// TIA Portal V20 export
FUNCTION_BLOCK "FB_Digital_Input"   // FB1, LAD
{ S7_Optimized_Access := 'TRUE' }
// stored: MemoryReserve 100, SetENOAutomatically false
   VAR_INPUT
      DI_Emergency_Stop_Release : Bool;
      DI_Sensor_Water_Fountain_Before_Entrace_Functional_Test_Spinner_Conveyor_Belt : Bool;
      DI_Sensor_Water_Fountain_Entrace_Functional_Test_Spinner_Conveyor_Belt : Bool;
      DI_Sensor_Water_Fountain_Entrace_Functional_Test_After_Spinner_Conveyor_Belt : Bool;
      DI_Trigger_Read_Serial_Number_Entrace_Functional_Test : Bool;
      DI_Sensor_Water_Fountain_Geting_Exit_Rework_Conveyor_Belt : Bool;
      DI_Button_Water_Fountain_Get_Exit_Rework_Conveyor_Belt : Bool;
      DI_Trigger_Read_Serial_Number_Exit_Functional_Test : Bool;
      DI_Sensor_Water_Fountain_Exit_Functional_Test_Spinner_Conveyor_Belt : Bool;
      DI_Sensor_Water_Fountain_Exit_Functional_Test_After_Spinner_Conveyor_Belt : Bool;
      DI_Sensor_Water_Fountain_Geting_Entrace_Rework_Conveyor_Belt_Start : Bool;
      DI_Sensor_Water_Fountain_Geting_Entrace_Rework_Conveyor_Belt_Finish : Bool;
      DI_Carousel_Frequency_Inverter_Fail : Bool;
      DI_Conveyor_Belt_Functional_Test_Inverter_Fail : Bool;
      DI_Selected_Voltage_220V : Bool;
      DI_Selected_Voltage_127V : Bool;
      DI_Sensor_Spinner_Entrace_Functional_Test_Position_Withdrawn : Bool;
      DI_Sensor_Spinner_Entrace_Functional_Test_Position_Advanced : Bool;
      DI_Sensor_Spinner_Exit_Functional_Test_Position_Withdrawn : Bool;
      DI_Sensor_Spinner_Exit_Functional_Test_Position_Advanced : Bool;
      DI_Digital_Input_20 : Bool;
      DI_Digital_Input_21 : Bool;
      DI_Digital_Input_22 : Bool;
      DI_Digital_Input_23 : Bool;
      DI_Digital_Input_24 : Bool;
      DI_Digital_Input_25 : Bool;
      DI_Digital_Input_26 : Bool;
      DI_Digital_Input_27 : Bool;
      DI_Digital_Input_28 : Bool;
      DI_Digital_Input_29 : Bool;
   END_VAR
   VAR_OUTPUT
      DB_Emergency_Stop_Release : Bool;
      DB_Sensor_Water_Fountain_Before_Entrace_Functional_Test_Spinner_Conveyor_Belt : Bool;
      DB_Sensor_Water_Fountain_Entrace_Functional_Test_Spinner_Conveyor_Belt : Bool;
      DB_Sensor_Water_Fountain_Entrace_Functional_Test_After_Spinner_Conveyor_Belt : Bool;
      DB_Trigger_Read_Serial_Number_Entrace_Functional_Test : Bool;
      DB_Sensor_Water_Fountain_Geting_Exit_Rework_Conveyor_Belt : Bool;
      DB_Button_Water_Fountain_Get_Exit_Rework_Conveyor_Belt : Bool;
      DB_Trigger_Read_Serial_Number_Exit_Functional_Test : Bool;
      DB_Sensor_Water_Fountain_Exit_Functional_Test_Spinner_Conveyor_Belt : Bool;
      DB_Sensor_Water_Fountain_Exit_Functional_Test_After_Spinner_Conveyor_Belt : Bool;
      DB_Sensor_Water_Fountain_Geting_Entrace_Rework_Conveyor_Belt_Start : Bool;
      DB_Sensor_Water_Fountain_Geting_Entrace_Rework_Conveyor_Belt_Finish : Bool;
      DB_Carousel_Frequency_Inverter_Fail : Bool;
      DB_Conveyor_Belt_Functional_Test_Inverter_Fail : Bool;
      DB_Selected_Voltage_220V : Bool;
      DB_Selected_Voltage_127V : Bool;
      DB_Sensor_Spinner_Entrace_Functional_Test_Position_Withdrawn : Bool;
      DB_Sensor_Spinner_Entrace_Functional_Test_Position_Advanced : Bool;
      DB_Sensor_Spinner_Exit_Functional_Test_Position_Withdrawn : Bool;
      DB_Sensor_Spinner_Exit_Functional_Test_Position_Advanced : Bool;
      DB_Digital_Input_20 : Bool;
      DB_Digital_Input_21 : Bool;
      DB_Digital_Input_22 : Bool;
      DB_Digital_Input_23 : Bool;
      DB_Digital_Input_24 : Bool;
      DB_Digital_Input_25 : Bool;
      DB_Digital_Input_26 : Bool;
      DB_Digital_Input_27 : Bool;
      DB_Digital_Input_28 : Bool;
      DB_Digital_Input_29 : Bool;
   END_VAR
BEGIN

REGION Network 1
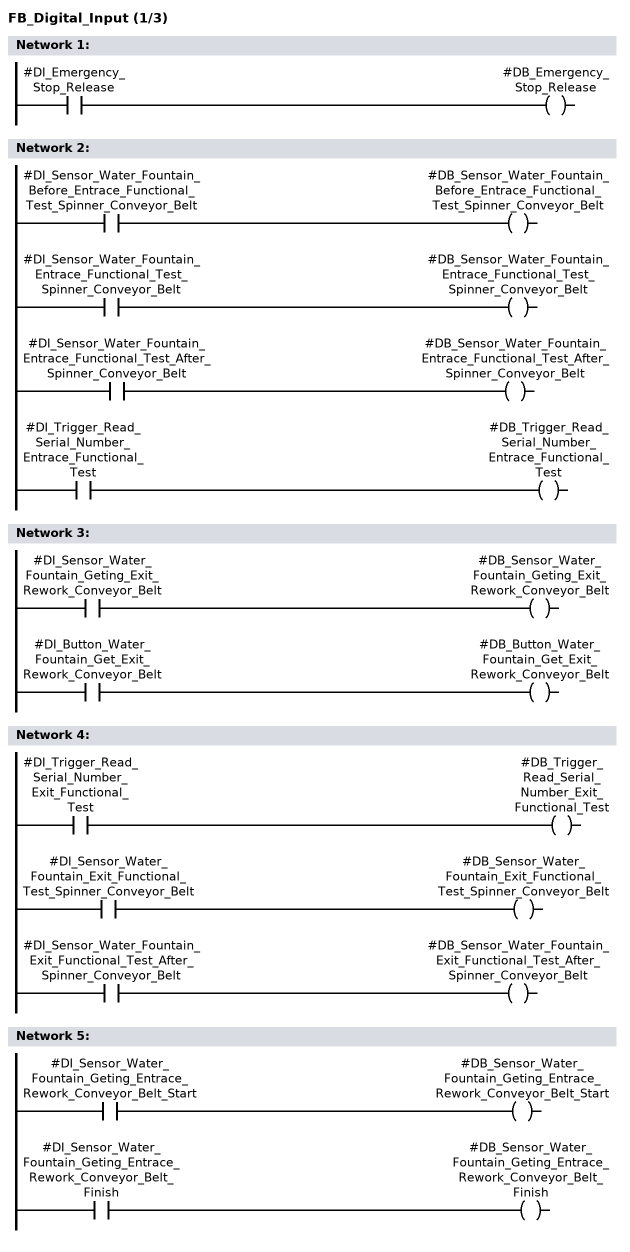
   RUNG wire#powerrail
      Contact( #DI_Emergency_Stop_Release )
      Coil( #DB_Emergency_Stop_Release )
   END_RUNG
   // the same network as SCL:
   #DB_Emergency_Stop_Release := #DI_Emergency_Stop_Release;
END_REGION

REGION Network 2
   RUNG wire#powerrail
      Contact( #DI_Sensor_Water_Fountain_Before_Entrace_Functional_Test_Spinner_Conveyor_Belt )
      Coil( #DB_Sensor_Water_Fountain_Before_Entrace_Functional_Test_Spinner_Conveyor_Belt )
   END_RUNG
   RUNG wire#powerrail
      Contact( #DI_Sensor_Water_Fountain_Entrace_Functional_Test_Spinner_Conveyor_Belt )
      Coil( #DB_Sensor_Water_Fountain_Entrace_Functional_Test_Spinner_Conveyor_Belt )
   END_RUNG
   RUNG wire#powerrail
      Contact( #DI_Sensor_Water_Fountain_Entrace_Functional_Test_After_Spinner_Conveyor_Belt )
      Coil( #DB_Sensor_Water_Fountain_Entrace_Functional_Test_After_Spinner_Conveyor_Belt )
   END_RUNG
   RUNG wire#powerrail
      Contact( #DI_Trigger_Read_Serial_Number_Entrace_Functional_Test )
      Coil( #DB_Trigger_Read_Serial_Number_Entrace_Functional_Test )
   END_RUNG
   // the same network as SCL:
   #DB_Sensor_Water_Fountain_Before_Entrace_Functional_Test_Spinner_Conveyor_Belt := #DI_Sensor_Water_Fountain_Before_Entrace_Functional_Test_Spinner_Conveyor_Belt;
   #DB_Sensor_Water_Fountain_Entrace_Functional_Test_Spinner_Conveyor_Belt := #DI_Sensor_Water_Fountain_Entrace_Functional_Test_Spinner_Conveyor_Belt;
   #DB_Sensor_Water_Fountain_Entrace_Functional_Test_After_Spinner_Conveyor_Belt := #DI_Sensor_Water_Fountain_Entrace_Functional_Test_After_Spinner_Conveyor_Belt;
   #DB_Trigger_Read_Serial_Number_Entrace_Functional_Test := #DI_Trigger_Read_Serial_Number_Entrace_Functional_Test;
END_REGION

REGION Network 3
   RUNG wire#powerrail
      Contact( #DI_Sensor_Water_Fountain_Geting_Exit_Rework_Conveyor_Belt )
      Coil( #DB_Sensor_Water_Fountain_Geting_Exit_Rework_Conveyor_Belt )
   END_RUNG
   RUNG wire#powerrail
      Contact( #DI_Button_Water_Fountain_Get_Exit_Rework_Conveyor_Belt )
      Coil( #DB_Button_Water_Fountain_Get_Exit_Rework_Conveyor_Belt )
   END_RUNG
   // the same network as SCL:
   #DB_Sensor_Water_Fountain_Geting_Exit_Rework_Conveyor_Belt := #DI_Sensor_Water_Fountain_Geting_Exit_Rework_Conveyor_Belt;
   #DB_Button_Water_Fountain_Get_Exit_Rework_Conveyor_Belt := #DI_Button_Water_Fountain_Get_Exit_Rework_Conveyor_Belt;
END_REGION

REGION Network 4
   RUNG wire#powerrail
      Contact( #DI_Trigger_Read_Serial_Number_Exit_Functional_Test )
      Coil( #DB_Trigger_Read_Serial_Number_Exit_Functional_Test )
   END_RUNG
   RUNG wire#powerrail
      Contact( #DI_Sensor_Water_Fountain_Exit_Functional_Test_Spinner_Conveyor_Belt )
      Coil( #DB_Sensor_Water_Fountain_Exit_Functional_Test_Spinner_Conveyor_Belt )
   END_RUNG
   RUNG wire#powerrail
      Contact( #DI_Sensor_Water_Fountain_Exit_Functional_Test_After_Spinner_Conveyor_Belt )
      Coil( #DB_Sensor_Water_Fountain_Exit_Functional_Test_After_Spinner_Conveyor_Belt )
   END_RUNG
   // the same network as SCL:
   #DB_Trigger_Read_Serial_Number_Exit_Functional_Test := #DI_Trigger_Read_Serial_Number_Exit_Functional_Test;
   #DB_Sensor_Water_Fountain_Exit_Functional_Test_Spinner_Conveyor_Belt := #DI_Sensor_Water_Fountain_Exit_Functional_Test_Spinner_Conveyor_Belt;
   #DB_Sensor_Water_Fountain_Exit_Functional_Test_After_Spinner_Conveyor_Belt := #DI_Sensor_Water_Fountain_Exit_Functional_Test_After_Spinner_Conveyor_Belt;
END_REGION

REGION Network 5
   RUNG wire#powerrail
      Contact( #DI_Sensor_Water_Fountain_Geting_Entrace_Rework_Conveyor_Belt_Start )
      Coil( #DB_Sensor_Water_Fountain_Geting_Entrace_Rework_Conveyor_Belt_Start )
   END_RUNG
   RUNG wire#powerrail
      Contact( #DI_Sensor_Water_Fountain_Geting_Entrace_Rework_Conveyor_Belt_Finish )
      Coil( #DB_Sensor_Water_Fountain_Geting_Entrace_Rework_Conveyor_Belt_Finish )
   END_RUNG
   // the same network as SCL:
   #DB_Sensor_Water_Fountain_Geting_Entrace_Rework_Conveyor_Belt_Start := #DI_Sensor_Water_Fountain_Geting_Entrace_Rework_Conveyor_Belt_Start;
   #DB_Sensor_Water_Fountain_Geting_Entrace_Rework_Conveyor_Belt_Finish := #DI_Sensor_Water_Fountain_Geting_Entrace_Rework_Conveyor_Belt_Finish;
END_REGION

REGION Network 6
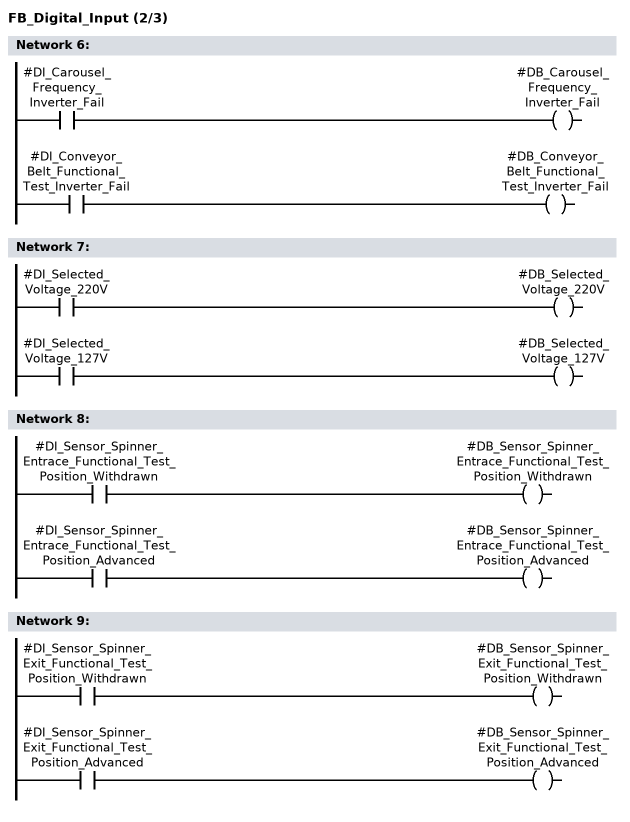
   RUNG wire#powerrail
      Contact( #DI_Carousel_Frequency_Inverter_Fail )
      Coil( #DB_Carousel_Frequency_Inverter_Fail )
   END_RUNG
   RUNG wire#powerrail
      Contact( #DI_Conveyor_Belt_Functional_Test_Inverter_Fail )
      Coil( #DB_Conveyor_Belt_Functional_Test_Inverter_Fail )
   END_RUNG
   // the same network as SCL:
   #DB_Carousel_Frequency_Inverter_Fail := #DI_Carousel_Frequency_Inverter_Fail;
   #DB_Conveyor_Belt_Functional_Test_Inverter_Fail := #DI_Conveyor_Belt_Functional_Test_Inverter_Fail;
END_REGION

REGION Network 7
   RUNG wire#powerrail
      Contact( #DI_Selected_Voltage_220V )
      Coil( #DB_Selected_Voltage_220V )
   END_RUNG
   RUNG wire#powerrail
      Contact( #DI_Selected_Voltage_127V )
      Coil( #DB_Selected_Voltage_127V )
   END_RUNG
   // the same network as SCL:
   #DB_Selected_Voltage_220V := #DI_Selected_Voltage_220V;
   #DB_Selected_Voltage_127V := #DI_Selected_Voltage_127V;
END_REGION

REGION Network 8
   RUNG wire#powerrail
      Contact( #DI_Sensor_Spinner_Entrace_Functional_Test_Position_Withdrawn )
      Coil( #DB_Sensor_Spinner_Entrace_Functional_Test_Position_Withdrawn )
   END_RUNG
   RUNG wire#powerrail
      Contact( #DI_Sensor_Spinner_Entrace_Functional_Test_Position_Advanced )
      Coil( #DB_Sensor_Spinner_Entrace_Functional_Test_Position_Advanced )
   END_RUNG
   // the same network as SCL:
   #DB_Sensor_Spinner_Entrace_Functional_Test_Position_Withdrawn := #DI_Sensor_Spinner_Entrace_Functional_Test_Position_Withdrawn;
   #DB_Sensor_Spinner_Entrace_Functional_Test_Position_Advanced := #DI_Sensor_Spinner_Entrace_Functional_Test_Position_Advanced;
END_REGION

REGION Network 9
   RUNG wire#powerrail
      Contact( #DI_Sensor_Spinner_Exit_Functional_Test_Position_Withdrawn )
      Coil( #DB_Sensor_Spinner_Exit_Functional_Test_Position_Withdrawn )
   END_RUNG
   RUNG wire#powerrail
      Contact( #DI_Sensor_Spinner_Exit_Functional_Test_Position_Advanced )
      Coil( #DB_Sensor_Spinner_Exit_Functional_Test_Position_Advanced )
   END_RUNG
   // the same network as SCL:
   #DB_Sensor_Spinner_Exit_Functional_Test_Position_Withdrawn := #DI_Sensor_Spinner_Exit_Functional_Test_Position_Withdrawn;
   #DB_Sensor_Spinner_Exit_Functional_Test_Position_Advanced := #DI_Sensor_Spinner_Exit_Functional_Test_Position_Advanced;
END_REGION

REGION Network 10
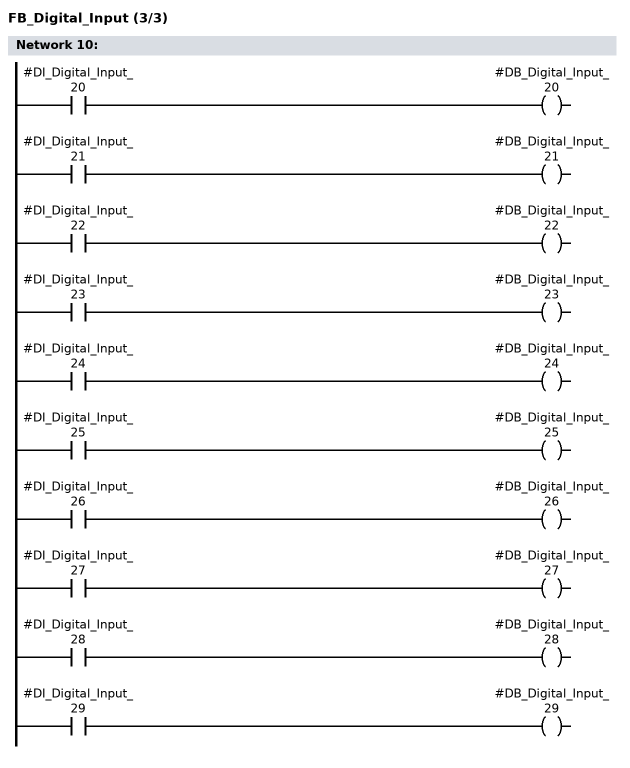
   RUNG wire#powerrail
      Contact( #DI_Digital_Input_20 )
      Coil( #DB_Digital_Input_20 )
   END_RUNG
   RUNG wire#powerrail
      Contact( #DI_Digital_Input_21 )
      Coil( #DB_Digital_Input_21 )
   END_RUNG
   RUNG wire#powerrail
      Contact( #DI_Digital_Input_22 )
      Coil( #DB_Digital_Input_22 )
   END_RUNG
   RUNG wire#powerrail
      Contact( #DI_Digital_Input_23 )
      Coil( #DB_Digital_Input_23 )
   END_RUNG
   RUNG wire#powerrail
      Contact( #DI_Digital_Input_24 )
      Coil( #DB_Digital_Input_24 )
   END_RUNG
   RUNG wire#powerrail
      Contact( #DI_Digital_Input_25 )
      Coil( #DB_Digital_Input_25 )
   END_RUNG
   RUNG wire#powerrail
      Contact( #DI_Digital_Input_26 )
      Coil( #DB_Digital_Input_26 )
   END_RUNG
   RUNG wire#powerrail
      Contact( #DI_Digital_Input_27 )
      Coil( #DB_Digital_Input_27 )
   END_RUNG
   RUNG wire#powerrail
      Contact( #DI_Digital_Input_28 )
      Coil( #DB_Digital_Input_28 )
   END_RUNG
   RUNG wire#powerrail
      Contact( #DI_Digital_Input_29 )
      Coil( #DB_Digital_Input_29 )
   END_RUNG
   // the same network as SCL:
   #DB_Digital_Input_20 := #DI_Digital_Input_20;
   #DB_Digital_Input_21 := #DI_Digital_Input_21;
   #DB_Digital_Input_22 := #DI_Digital_Input_22;
   #DB_Digital_Input_23 := #DI_Digital_Input_23;
   #DB_Digital_Input_24 := #DI_Digital_Input_24;
   #DB_Digital_Input_25 := #DI_Digital_Input_25;
   #DB_Digital_Input_26 := #DI_Digital_Input_26;
   #DB_Digital_Input_27 := #DI_Digital_Input_27;
   #DB_Digital_Input_28 := #DI_Digital_Input_28;
   #DB_Digital_Input_29 := #DI_Digital_Input_29;
END_REGION
END_FUNCTION_BLOCK
